// TIA Portal V17 export
// export: Created 2024-09-02T12:50:18.0928197Z, ExportSetting WithDefaults, DisplayName Totally Integrated Automation Portal, DisplayVersion V17, DisplayName TIA Portal Openness, DisplayVersion V17, DisplayName TIA Portal Version Control Interface, DisplayVersion V17, DisplayName STEP 7 Professional, DisplayVersion V17, DisplayName STEP 7 Safety, DisplayVersion V17, DisplayName WinCC Professional, DisplayVersion V17
FUNCTION_BLOCK "LTLL_Main_HMI_OP70"   // FB3, LAD
TITLE = LTLL_HMILite
{ S7_Optimized_Access := 'TRUE' }
AUTHOR : Siemens
FAMILY : HMI_Lite
NAME : LTLL_HMILite
VERSION : 8.10
// stored: AutoNumber true, IsIECCheckEnabled false, IsRetainMemResEnabled false, MemoryReserve 100, SetENOAutomatically false, UDAEnableTagReadback false
   VAR
      instLTLL_Basic { S7_SetPoint := 'True'} : "LTLL_Basic";
      instLTLL_Manual { S7_SetPoint := 'True'} : "LTLL_Manual";
      instLTLL_ManualGraph { S7_SetPoint := 'True'} : "LTLL_ManualGraph";
      instLTLL_Sinamics { S7_SetPoint := 'True'} : "LTLL_Sinamics";
      instLTLL_Motorstarter { S7_SetPoint := 'True'} : "LTLL_Motorstarter";
      instLTLL_RFID { S7_SetPoint := 'True'} : "LTLL_RFID";
      instLTLL_Cycletime_1 { S7_SetPoint := 'True'} : "LTLL_Cycletime";
      instLTLL_Cycletime { S7_SetPoint := 'True'} : "LTLL_Cycletime";
      instLTLL_Counter { S7_SetPoint := 'True'} : "LTLL_Counter";
      instLTLL_PLCSystemData { S7_SetPoint := 'True'} : "LTLL_PLCSystemData";
      instLTLL_Eks { S7_SetPoint := 'True'} : "LTLL_Eks";
   END_VAR
   VAR_TEMP
      tempBasicRetRDSysT : Int;
      tempBasicStatusRDREC : DWord;
      tempBasicStatus : Word;
      tempBasicErrID : Word;
      tempManualStatus : Word;
      tempManualErrID : Word;
      tempManualGraphStatus : Word;
      tempManualGraphErrID : Word;
      tempSinamicsBusy : Bool;
      tempSinamicsStatus : Word;
      tempSinamicsErrID : Word;
      tempSinamicsWrRecStatus : DWord;
      tempSinamicsRdRecStatus : DWord;
      tempMotorstarterBusy : Bool;
      tempMotorstarterRdRec1Status : DWord;
      tempMotorstarterRdRec2Status : DWord;
      tempMotorstarterErrID : Word;
      tempMotorstarterStatus : Word;
      tempRfidStatus : Word;
      tempRfidErrID : Word;
      tempPlcSystemDataStatus : Word;
      tempPlcSystemDataStatusGetImData : Word;
      tempPlcSystemDataErrID : Word;
      tempCounter1Status : Word;
      tempCounter1ErrID : Word;
      tempCycletime1Status : Word;
      tempCycletime1ErrID : Word;
      tempEksProtectionLevel : Int;
      tempEksChecksumNOK : Bool;
      tempEksDateNOK : Bool;
      tempEkscostCenterNOK : Bool;
      tempEksKeyInvalidLess30Days : Bool;
      tempEksAdapterReady : Bool;
      tempEksKeyDetected : Bool;
      tempSchichtReset : Bool;
      tempTagReset : Bool;
      tempZeiger : Int;
      tempAnzGesamt : Int;
      tempAnzNio : Int;
      Cycle_Time_Index : Int;
      t_i : Int;
   END_VAR
   VAR_TEMP   // added for the SCL form of the ladder/FBD networks
      _w1 : Bool;
      _w2 : Bool;
      _w3 : Bool;
   END_VAR
BEGIN

REGION Network 1: Call HMI Lite Basic / Aufruf HMI Lite Basic
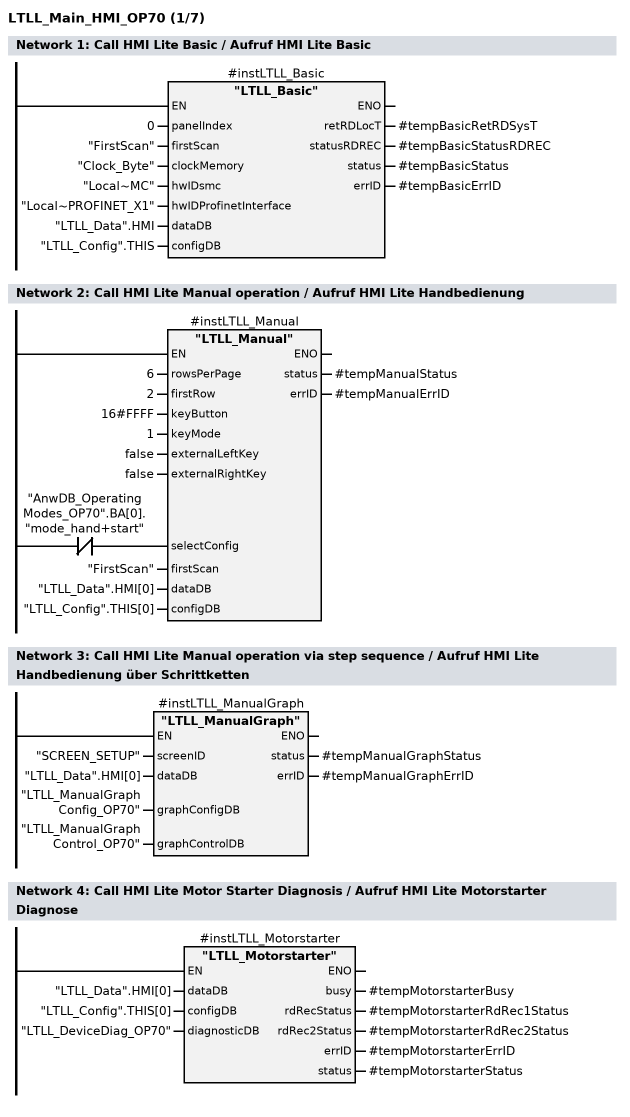
   RUNG wire#powerrail
      #instLTLL_Basic(panelIndex := 0, firstScan := "FirstScan", clockMemory := "Clock_Byte", hwIDsmc := "Local~MC", hwIDProfinetInterface := "Local~PROFINET_X1", dataDB := "LTLL_Data".HMI, configDB := "LTLL_Config".THIS, retRDLocT => #tempBasicRetRDSysT, statusRDREC => #tempBasicStatusRDREC, status => #tempBasicStatus, errID => #tempBasicErrID)
   END_RUNG
   // the same network as SCL:
   #instLTLL_Basic(panelIndex := 0,   // "LTLL_Basic"
                   firstScan := "FirstScan",
                   clockMemory := "Clock_Byte",
                   hwIDsmc := "Local~MC",
                   hwIDProfinetInterface := "Local~PROFINET_X1",
                   dataDB := "LTLL_Data".HMI,
                   configDB := "LTLL_Config".THIS,
                   retRDLocT => #tempBasicRetRDSysT,
                   statusRDREC => #tempBasicStatusRDREC,
                   status => #tempBasicStatus,
                   errID => #tempBasicErrID);
END_REGION

REGION Network 2: Call HMI Lite Manual operation / Aufruf HMI Lite Handbedienung
   RUNG wire#powerrail
      #instLTLL_Manual(selectConfig := wire#w1, rowsPerPage := 6, firstRow := 2, keyButton := 16#FFFF, keyMode := 1, externalLeftKey := false, externalRightKey := false, firstScan := "FirstScan", dataDB := "LTLL_Data".HMI[0], configDB := "LTLL_Config".THIS[0], status => #tempManualStatus, errID => #tempManualErrID)
   END_RUNG
   RUNG wire#powerrail
      I_Contact( "AnwDB_OperatingModes_OP70".BA[0]."mode_hand+start" )
   END_RUNG wire#w1
   // the same network as SCL:
   #instLTLL_Manual(rowsPerPage := 6,   // "LTLL_Manual"
                    firstRow := 2,
                    keyButton := 16#FFFF,
                    keyMode := 1,
                    externalLeftKey := false,
                    externalRightKey := false,
                    selectConfig := NOT "AnwDB_OperatingModes_OP70".BA[0]."mode_hand+start",
                    firstScan := "FirstScan",
                    dataDB := "LTLL_Data".HMI[0],
                    configDB := "LTLL_Config".THIS[0],
                    status => #tempManualStatus,
                    errID => #tempManualErrID);
END_REGION

REGION Network 3: Call HMI Lite Manual operation via step sequence / Aufruf HMI Lite Handbedienung über Schrittketten
   RUNG wire#powerrail
      #instLTLL_ManualGraph(screenID := "SCREEN_SETUP", dataDB := "LTLL_Data".HMI[0], graphConfigDB := "LTLL_ManualGraphConfig_OP70", graphControlDB := "LTLL_ManualGraphControl_OP70", status => #tempManualGraphStatus, errID => #tempManualGraphErrID)
   END_RUNG
   // the same network as SCL:
   #instLTLL_ManualGraph(screenID := "SCREEN_SETUP",   // "LTLL_ManualGraph"
                         dataDB := "LTLL_Data".HMI[0],
                         graphConfigDB := "LTLL_ManualGraphConfig_OP70",
                         graphControlDB := "LTLL_ManualGraphControl_OP70",
                         status => #tempManualGraphStatus,
                         errID => #tempManualGraphErrID);
END_REGION

REGION Network 4: Call HMI Lite Motor Starter Diagnosis / Aufruf HMI Lite Motorstarter Diagnose
   RUNG wire#powerrail
      #instLTLL_Motorstarter(dataDB := "LTLL_Data".HMI[0], configDB := "LTLL_Config".THIS[0], diagnosticDB := "LTLL_DeviceDiag_OP70", busy => #tempMotorstarterBusy, rdRecStatus => #tempMotorstarterRdRec1Status, rdRec2Status => #tempMotorstarterRdRec2Status, errID => #tempMotorstarterErrID, status => #tempMotorstarterStatus)
   END_RUNG
   // the same network as SCL:
   #instLTLL_Motorstarter(dataDB := "LTLL_Data".HMI[0],   // "LTLL_Motorstarter"
                          configDB := "LTLL_Config".THIS[0],
                          diagnosticDB := "LTLL_DeviceDiag_OP70",
                          busy => #tempMotorstarterBusy,
                          rdRecStatus => #tempMotorstarterRdRec1Status,
                          rdRec2Status => #tempMotorstarterRdRec2Status,
                          errID => #tempMotorstarterErrID,
                          status => #tempMotorstarterStatus);
END_REGION

REGION Network 5: Call the HMI Lite RFID Diagnostics / Auruf der HMI Lite RFID Diagnose
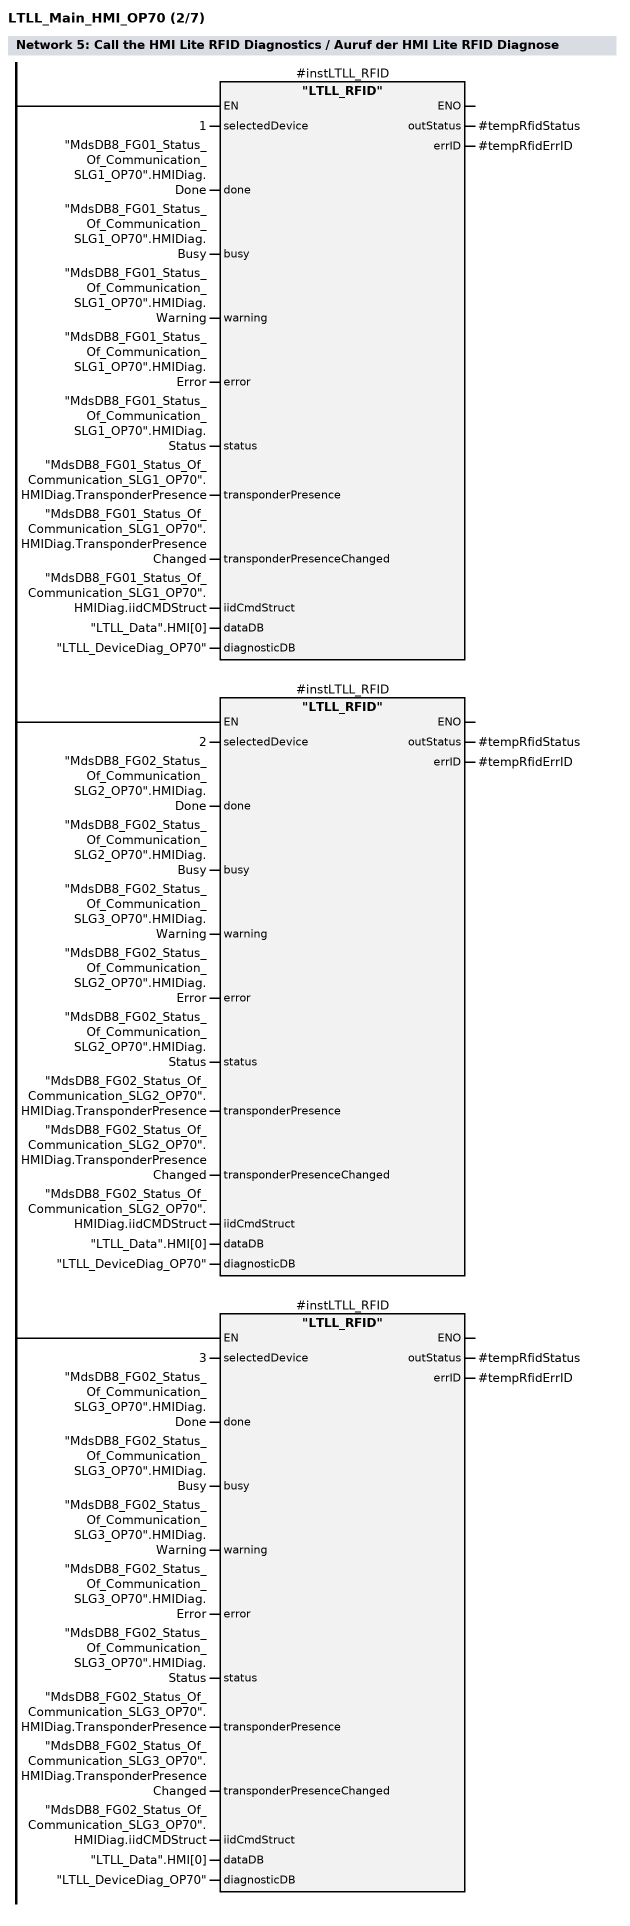
   RUNG wire#powerrail
      #instLTLL_RFID(selectedDevice := 1, done := "MdsDB8_FG01_Status_Of_Communication_SLG1_OP70".HMIDiag.Done, busy := "MdsDB8_FG01_Status_Of_Communication_SLG1_OP70".HMIDiag.Busy, warning := "MdsDB8_FG01_Status_Of_Communication_SLG1_OP70".HMIDiag.Warning, error := "MdsDB8_FG01_Status_Of_Communication_SLG1_OP70".HMIDiag.Error, status := "MdsDB8_FG01_Status_Of_Communication_SLG1_OP70".HMIDiag.Status, transponderPresence := "MdsDB8_FG01_Status_Of_Communication_SLG1_OP70".HMIDiag.TransponderPresence, transponderPresenceChanged := "MdsDB8_FG01_Status_Of_Communication_SLG1_OP70".HMIDiag.TransponderPresenceChanged, iidCmdStruct := "MdsDB8_FG01_Status_Of_Communication_SLG1_OP70".HMIDiag.iidCMDStruct, dataDB := "LTLL_Data".HMI[0], diagnosticDB := "LTLL_DeviceDiag_OP70", outStatus => #tempRfidStatus, errID => #tempRfidErrID)
   END_RUNG
   RUNG wire#powerrail
      #instLTLL_RFID(selectedDevice := 2, done := "MdsDB8_FG02_Status_Of_Communication_SLG2_OP70".HMIDiag.Done, busy := "MdsDB8_FG02_Status_Of_Communication_SLG2_OP70".HMIDiag.Busy, warning := "MdsDB8_FG02_Status_Of_Communication_SLG3_OP70".HMIDiag.Warning, error := "MdsDB8_FG02_Status_Of_Communication_SLG2_OP70".HMIDiag.Error, status := "MdsDB8_FG02_Status_Of_Communication_SLG2_OP70".HMIDiag.Status, transponderPresence := "MdsDB8_FG02_Status_Of_Communication_SLG2_OP70".HMIDiag.TransponderPresence, transponderPresenceChanged := "MdsDB8_FG02_Status_Of_Communication_SLG2_OP70".HMIDiag.TransponderPresenceChanged, iidCmdStruct := "MdsDB8_FG02_Status_Of_Communication_SLG2_OP70".HMIDiag.iidCMDStruct, dataDB := "LTLL_Data".HMI[0], diagnosticDB := "LTLL_DeviceDiag_OP70", outStatus => #tempRfidStatus, errID => #tempRfidErrID)
   END_RUNG
   RUNG wire#powerrail
      #instLTLL_RFID(selectedDevice := 3, done := "MdsDB8_FG02_Status_Of_Communication_SLG3_OP70".HMIDiag.Done, busy := "MdsDB8_FG02_Status_Of_Communication_SLG3_OP70".HMIDiag.Busy, warning := "MdsDB8_FG02_Status_Of_Communication_SLG3_OP70".HMIDiag.Warning, error := "MdsDB8_FG02_Status_Of_Communication_SLG3_OP70".HMIDiag.Error, status := "MdsDB8_FG02_Status_Of_Communication_SLG3_OP70".HMIDiag.Status, transponderPresence := "MdsDB8_FG02_Status_Of_Communication_SLG3_OP70".HMIDiag.TransponderPresence, transponderPresenceChanged := "MdsDB8_FG02_Status_Of_Communication_SLG3_OP70".HMIDiag.TransponderPresenceChanged, iidCmdStruct := "MdsDB8_FG02_Status_Of_Communication_SLG3_OP70".HMIDiag.iidCMDStruct, dataDB := "LTLL_Data".HMI[0], diagnosticDB := "LTLL_DeviceDiag_OP70", outStatus => #tempRfidStatus, errID => #tempRfidErrID)
   END_RUNG
   // the same network as SCL:
   #instLTLL_RFID(selectedDevice := 1,   // "LTLL_RFID"
                  done := "MdsDB8_FG01_Status_Of_Communication_SLG1_OP70".HMIDiag.Done,
                  busy := "MdsDB8_FG01_Status_Of_Communication_SLG1_OP70".HMIDiag.Busy,
                  warning := "MdsDB8_FG01_Status_Of_Communication_SLG1_OP70".HMIDiag.Warning,
                  error := "MdsDB8_FG01_Status_Of_Communication_SLG1_OP70".HMIDiag.Error,
                  status := "MdsDB8_FG01_Status_Of_Communication_SLG1_OP70".HMIDiag.Status,
                  transponderPresence := "MdsDB8_FG01_Status_Of_Communication_SLG1_OP70".HMIDiag.TransponderPresence,
                  transponderPresenceChanged := "MdsDB8_FG01_Status_Of_Communication_SLG1_OP70".HMIDiag.TransponderPresenceChanged,
                  iidCmdStruct := "MdsDB8_FG01_Status_Of_Communication_SLG1_OP70".HMIDiag.iidCMDStruct,
                  dataDB := "LTLL_Data".HMI[0],
                  diagnosticDB := "LTLL_DeviceDiag_OP70",
                  outStatus => #tempRfidStatus,
                  errID => #tempRfidErrID);
   #instLTLL_RFID(selectedDevice := 2,   // "LTLL_RFID"
                  done := "MdsDB8_FG02_Status_Of_Communication_SLG2_OP70".HMIDiag.Done,
                  busy := "MdsDB8_FG02_Status_Of_Communication_SLG2_OP70".HMIDiag.Busy,
                  warning := "MdsDB8_FG02_Status_Of_Communication_SLG3_OP70".HMIDiag.Warning,
                  error := "MdsDB8_FG02_Status_Of_Communication_SLG2_OP70".HMIDiag.Error,
                  status := "MdsDB8_FG02_Status_Of_Communication_SLG2_OP70".HMIDiag.Status,
                  transponderPresence := "MdsDB8_FG02_Status_Of_Communication_SLG2_OP70".HMIDiag.TransponderPresence,
                  transponderPresenceChanged := "MdsDB8_FG02_Status_Of_Communication_SLG2_OP70".HMIDiag.TransponderPresenceChanged,
                  iidCmdStruct := "MdsDB8_FG02_Status_Of_Communication_SLG2_OP70".HMIDiag.iidCMDStruct,
                  dataDB := "LTLL_Data".HMI[0],
                  diagnosticDB := "LTLL_DeviceDiag_OP70",
                  outStatus => #tempRfidStatus,
                  errID => #tempRfidErrID);
   #instLTLL_RFID(selectedDevice := 3,   // "LTLL_RFID"
                  done := "MdsDB8_FG02_Status_Of_Communication_SLG3_OP70".HMIDiag.Done,
                  busy := "MdsDB8_FG02_Status_Of_Communication_SLG3_OP70".HMIDiag.Busy,
                  warning := "MdsDB8_FG02_Status_Of_Communication_SLG3_OP70".HMIDiag.Warning,
                  error := "MdsDB8_FG02_Status_Of_Communication_SLG3_OP70".HMIDiag.Error,
                  status := "MdsDB8_FG02_Status_Of_Communication_SLG3_OP70".HMIDiag.Status,
                  transponderPresence := "MdsDB8_FG02_Status_Of_Communication_SLG3_OP70".HMIDiag.TransponderPresence,
                  transponderPresenceChanged := "MdsDB8_FG02_Status_Of_Communication_SLG3_OP70".HMIDiag.TransponderPresenceChanged,
                  iidCmdStruct := "MdsDB8_FG02_Status_Of_Communication_SLG3_OP70".HMIDiag.iidCMDStruct,
                  dataDB := "LTLL_Data".HMI[0],
                  diagnosticDB := "LTLL_DeviceDiag_OP70",
                  outStatus => #tempRfidStatus,
                  errID => #tempRfidErrID);
END_REGION

REGION Network 6: Call HMI Lite PLC system data / Aufruf HMI Lite PLC Systemdaten
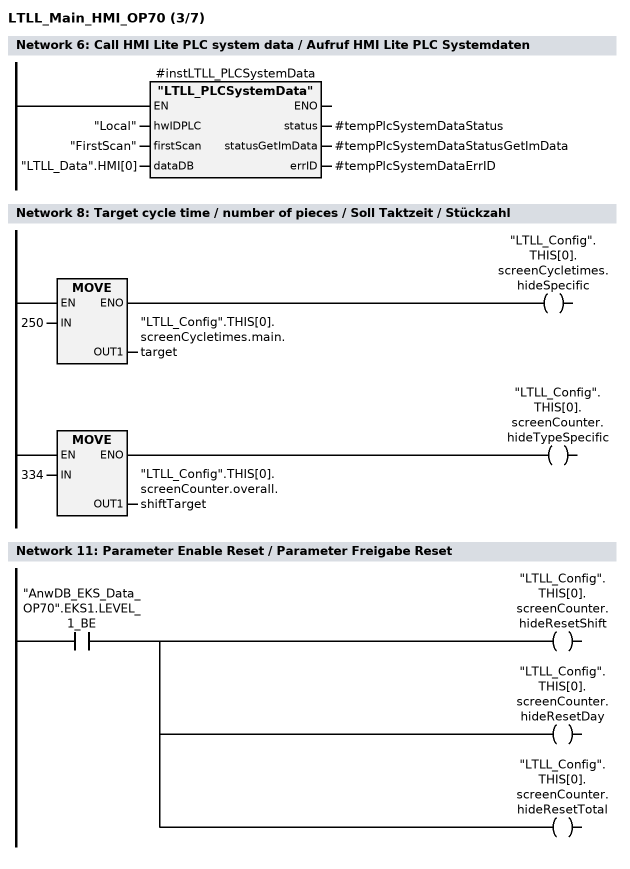
   RUNG wire#powerrail
      #instLTLL_PLCSystemData(hwIDPLC := "Local", firstScan := "FirstScan", dataDB := "LTLL_Data".HMI[0], status => #tempPlcSystemDataStatus, statusGetImData => #tempPlcSystemDataStatusGetImData, errID => #tempPlcSystemDataErrID)
   END_RUNG
   // the same network as SCL:
   #instLTLL_PLCSystemData(hwIDPLC := "Local",   // "LTLL_PLCSystemData"
                           firstScan := "FirstScan",
                           dataDB := "LTLL_Data".HMI[0],
                           status => #tempPlcSystemDataStatus,
                           statusGetImData => #tempPlcSystemDataStatusGetImData,
                           errID => #tempPlcSystemDataErrID);
END_REGION

REGION Network 7: Call HMI Lite Safety Diagnosis / Aufruf HMI Lite Safety Diagnose
END_REGION

REGION Network 8: Target cycle time / number of pieces / Soll Taktzeit / Stückzahl
   RUNG wire#powerrail
      Move(in := 250, out1 => "LTLL_Config".THIS[0].screenCycletimes.main.target)
      Coil( "LTLL_Config".THIS[0].screenCycletimes.hideSpecific )
   END_RUNG
   RUNG wire#powerrail
      Move(in := 334, out1 => "LTLL_Config".THIS[0].screenCounter.overall.shiftTarget)
      Coil( "LTLL_Config".THIS[0].screenCounter.hideTypeSpecific )
   END_RUNG
   // the same network as SCL:
   "LTLL_Config".THIS[0].screenCycletimes.main.target := 250;
   "LTLL_Config".THIS[0].screenCycletimes.hideSpecific := TRUE;
   "LTLL_Config".THIS[0].screenCounter.overall.shiftTarget := 334;
   "LTLL_Config".THIS[0].screenCounter.hideTypeSpecific := TRUE;
END_REGION

REGION Network 9 (SCL): Target cycle time Sub
   FOR #t_i := 0 TO 14 DO
       "LTLL_Config".THIS[0].screenCycletimes.sub.target[#t_i] := "LTLL_Config".THIS[0].screenCycletimes.main.target;

   END_FOR;
END_REGION

REGION Network 10 (SCL): Specific quantity Target quantity / Stückzahl spezifisch Soll
   FOR #tempZeiger := 0 TO 31 DO
       "LTLL_CounterData_OP70".specific[#tempZeiger].config.shiftTarget := 0;
   END_FOR;
END_REGION

REGION Network 11: Parameter Enable Reset / Parameter Freigabe Reset
   RUNG wire#powerrail
      Contact( "AnwDB_EKS_Data_OP70".EKS1.LEVEL_1_BE )
      wire#w1
      Coil( "LTLL_Config".THIS[0].screenCounter.hideResetShift )
   END_RUNG
   RUNG wire#w1
      Coil( "LTLL_Config".THIS[0].screenCounter.hideResetDay )
   END_RUNG
   RUNG wire#w1
      Coil( "LTLL_Config".THIS[0].screenCounter.hideResetTotal )
   END_RUNG
   // the same network as SCL:
   "LTLL_Config".THIS[0].screenCounter.hideResetShift := "AnwDB_EKS_Data_OP70".EKS1.LEVEL_1_BE;
   "LTLL_Config".THIS[0].screenCounter.hideResetDay := "AnwDB_EKS_Data_OP70".EKS1.LEVEL_1_BE;
   "LTLL_Config".THIS[0].screenCounter.hideResetTotal := "AnwDB_EKS_Data_OP70".EKS1.LEVEL_1_BE;
END_REGION

REGION Network 12: Quantity Reset / Stückzahl Reset
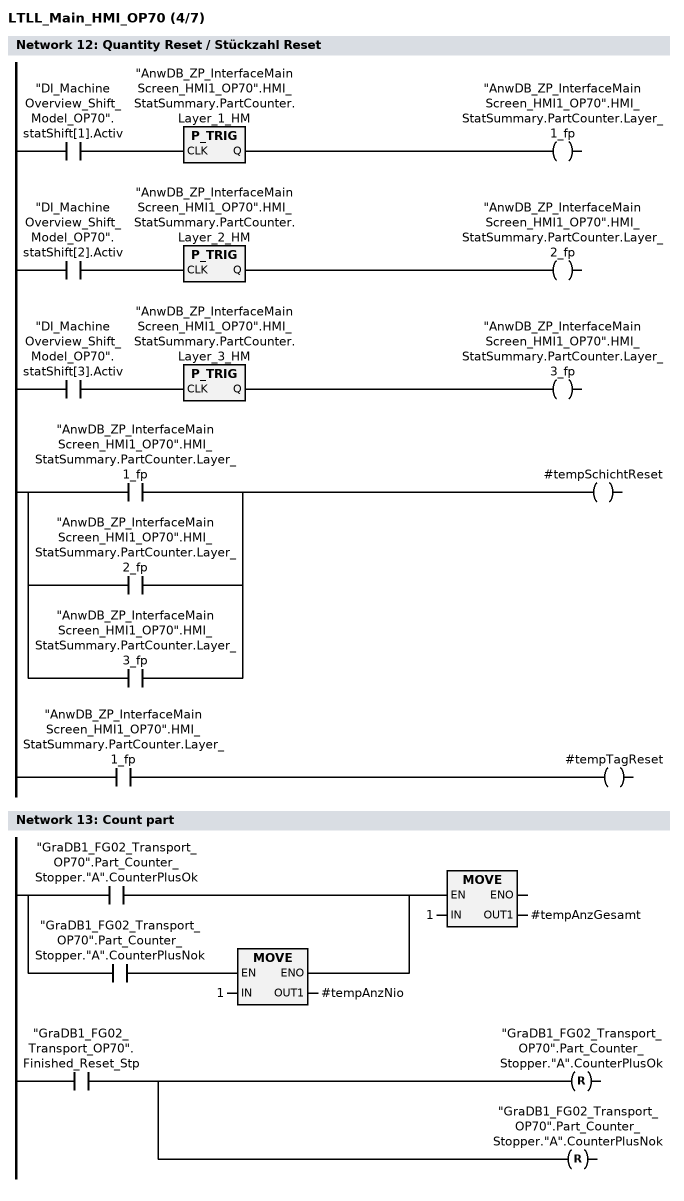
   RUNG wire#powerrail
      Contact( "DI_MachineOverview_Shift_Model_OP70".statShift[1].Activ )
      P_Trig( "AnwDB_ZP_InterfaceMainScreen_HMI1_OP70".HMI_StatSummary.PartCounter.Layer_1_HM )
      Coil( "AnwDB_ZP_InterfaceMainScreen_HMI1_OP70".HMI_StatSummary.PartCounter.Layer_1_fp )
   END_RUNG
   RUNG wire#powerrail
      Contact( "DI_MachineOverview_Shift_Model_OP70".statShift[2].Activ )
      P_Trig( "AnwDB_ZP_InterfaceMainScreen_HMI1_OP70".HMI_StatSummary.PartCounter.Layer_2_HM )
      Coil( "AnwDB_ZP_InterfaceMainScreen_HMI1_OP70".HMI_StatSummary.PartCounter.Layer_2_fp )
   END_RUNG
   RUNG wire#powerrail
      Contact( "DI_MachineOverview_Shift_Model_OP70".statShift[3].Activ )
      P_Trig( "AnwDB_ZP_InterfaceMainScreen_HMI1_OP70".HMI_StatSummary.PartCounter.Layer_3_HM )
      Coil( "AnwDB_ZP_InterfaceMainScreen_HMI1_OP70".HMI_StatSummary.PartCounter.Layer_3_fp )
   END_RUNG
   RUNG wire#powerrail
      Contact( "AnwDB_ZP_InterfaceMainScreen_HMI1_OP70".HMI_StatSummary.PartCounter.Layer_1_fp )
      wire#w1
      Coil( #tempSchichtReset )
   END_RUNG
   RUNG wire#powerrail
      Contact( "AnwDB_ZP_InterfaceMainScreen_HMI1_OP70".HMI_StatSummary.PartCounter.Layer_2_fp )
   END_RUNG wire#w1
   RUNG wire#powerrail
      Contact( "AnwDB_ZP_InterfaceMainScreen_HMI1_OP70".HMI_StatSummary.PartCounter.Layer_3_fp )
   END_RUNG wire#w1
   RUNG wire#powerrail
      Contact( "AnwDB_ZP_InterfaceMainScreen_HMI1_OP70".HMI_StatSummary.PartCounter.Layer_1_fp )
      Coil( #tempTagReset )
   END_RUNG
   // the same network as SCL:
   #_w1 := "DI_MachineOverview_Shift_Model_OP70".statShift[1].Activ AND NOT "AnwDB_ZP_InterfaceMainScreen_HMI1_OP70".HMI_StatSummary.PartCounter.Layer_1_HM;   // rising edge
   "AnwDB_ZP_InterfaceMainScreen_HMI1_OP70".HMI_StatSummary.PartCounter.Layer_1_HM := "DI_MachineOverview_Shift_Model_OP70".statShift[1].Activ;
   "AnwDB_ZP_InterfaceMainScreen_HMI1_OP70".HMI_StatSummary.PartCounter.Layer_1_fp := #_w1;
   #_w2 := "DI_MachineOverview_Shift_Model_OP70".statShift[2].Activ AND NOT "AnwDB_ZP_InterfaceMainScreen_HMI1_OP70".HMI_StatSummary.PartCounter.Layer_2_HM;   // rising edge
   "AnwDB_ZP_InterfaceMainScreen_HMI1_OP70".HMI_StatSummary.PartCounter.Layer_2_HM := "DI_MachineOverview_Shift_Model_OP70".statShift[2].Activ;
   "AnwDB_ZP_InterfaceMainScreen_HMI1_OP70".HMI_StatSummary.PartCounter.Layer_2_fp := #_w2;
   #_w3 := "DI_MachineOverview_Shift_Model_OP70".statShift[3].Activ AND NOT "AnwDB_ZP_InterfaceMainScreen_HMI1_OP70".HMI_StatSummary.PartCounter.Layer_3_HM;   // rising edge
   "AnwDB_ZP_InterfaceMainScreen_HMI1_OP70".HMI_StatSummary.PartCounter.Layer_3_HM := "DI_MachineOverview_Shift_Model_OP70".statShift[3].Activ;
   "AnwDB_ZP_InterfaceMainScreen_HMI1_OP70".HMI_StatSummary.PartCounter.Layer_3_fp := #_w3;
   #tempSchichtReset := "AnwDB_ZP_InterfaceMainScreen_HMI1_OP70".HMI_StatSummary.PartCounter.Layer_1_fp OR "AnwDB_ZP_InterfaceMainScreen_HMI1_OP70".HMI_StatSummary.PartCounter.Layer_2_fp OR "AnwDB_ZP_InterfaceMainScreen_HMI1_OP70".HMI_StatSummary.PartCounter.Layer_3_fp;
   #tempTagReset := "AnwDB_ZP_InterfaceMainScreen_HMI1_OP70".HMI_StatSummary.PartCounter.Layer_1_fp;
END_REGION

REGION Network 13: Count part
   RUNG wire#powerrail
      Contact( "GraDB1_FG02_Transport_OP70".Part_Counter_Stopper."A".CounterPlusOk )
      wire#w1
      Move(in := 1, out1 => #tempAnzGesamt)
   END_RUNG
   RUNG wire#powerrail
      Contact( "GraDB1_FG02_Transport_OP70".Part_Counter_Stopper."A".CounterPlusNok )
      Move(in := 1, out1 => #tempAnzNio)
   END_RUNG wire#w1
   RUNG wire#powerrail
      Contact( "GraDB1_FG02_Transport_OP70".Finished_Reset_Stp )
      wire#w2
      R_Coil( "GraDB1_FG02_Transport_OP70".Part_Counter_Stopper."A".CounterPlusOk )
   END_RUNG
   RUNG wire#w2
      R_Coil( "GraDB1_FG02_Transport_OP70".Part_Counter_Stopper."A".CounterPlusNok )
   END_RUNG
   // the same network as SCL:
   IF "GraDB1_FG02_Transport_OP70".Part_Counter_Stopper."A".CounterPlusNok THEN #tempAnzNio := 1; END_IF;
   IF "GraDB1_FG02_Transport_OP70".Part_Counter_Stopper."A".CounterPlusOk OR "GraDB1_FG02_Transport_OP70".Part_Counter_Stopper."A".CounterPlusNok THEN
       #tempAnzGesamt := 1;
   END_IF;
   IF "GraDB1_FG02_Transport_OP70".Finished_Reset_Stp THEN
       "GraDB1_FG02_Transport_OP70".Part_Counter_Stopper."A".CounterPlusOk := FALSE;
       "GraDB1_FG02_Transport_OP70".Part_Counter_Stopper."A".CounterPlusNok := FALSE;
   END_IF;
END_REGION

REGION Network 14: Call HMI Lite piece counter / Aufruf HMI Lite Stückzähler
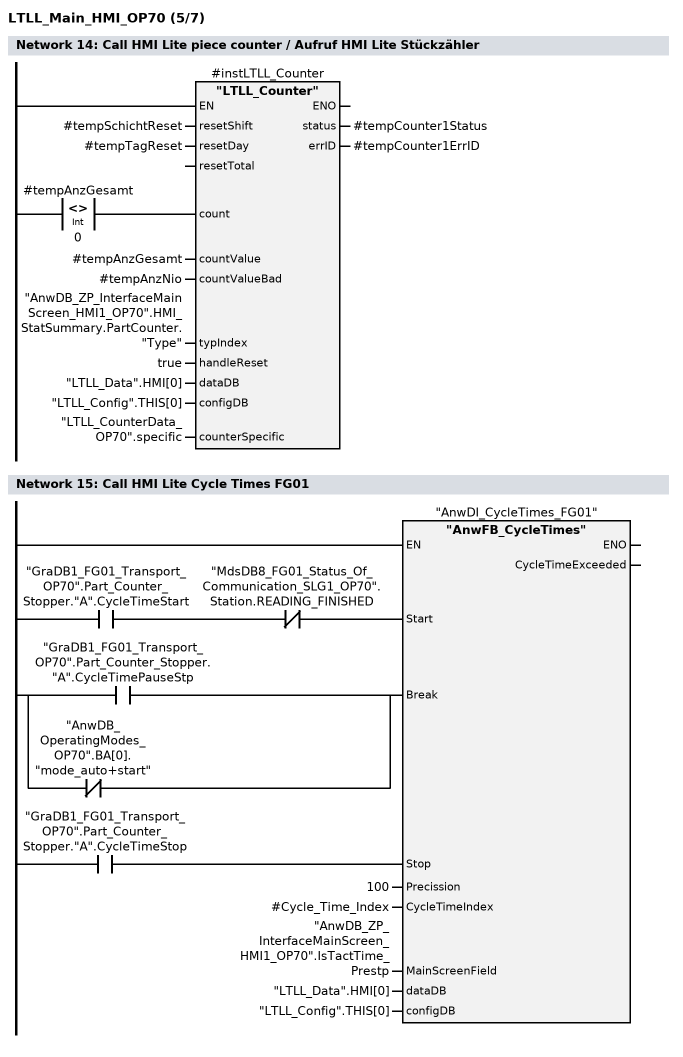
   RUNG wire#powerrail
      #instLTLL_Counter(count := wire#w1, resetShift := #tempSchichtReset, resetDay := #tempTagReset, resetTotal :=, countValue := #tempAnzGesamt, countValueBad := #tempAnzNio, typIndex := "AnwDB_ZP_InterfaceMainScreen_HMI1_OP70".HMI_StatSummary.PartCounter."Type", handleReset := true, dataDB := "LTLL_Data".HMI[0], configDB := "LTLL_Config".THIS[0], counterSpecific := "LTLL_CounterData_OP70".specific, status => #tempCounter1Status, errID => #tempCounter1ErrID)
   END_RUNG
   RUNG wire#powerrail
      { S7_Templates := "SrcType := Int" } NE_Contact(in1 := #tempAnzGesamt, in2 := 0)
   END_RUNG wire#w1
   // the same network as SCL:
   #instLTLL_Counter(resetShift := #tempSchichtReset,   // "LTLL_Counter"
                     resetDay := #tempTagReset,
                     count := #tempAnzGesamt <> 0,
                     countValue := #tempAnzGesamt,
                     countValueBad := #tempAnzNio,
                     typIndex := "AnwDB_ZP_InterfaceMainScreen_HMI1_OP70".HMI_StatSummary.PartCounter."Type",
                     handleReset := true,
                     dataDB := "LTLL_Data".HMI[0],
                     configDB := "LTLL_Config".THIS[0],
                     counterSpecific := "LTLL_CounterData_OP70".specific,
                     status => #tempCounter1Status,
                     errID => #tempCounter1ErrID);
END_REGION

REGION Network 15: Call HMI Lite Cycle Times FG01
   RUNG wire#powerrail
      "AnwDI_CycleTimes_FG01"(Start := wire#w1, Break := wire#w2, Stop := wire#w3, Precission := 100, CycleTimeIndex := #Cycle_Time_Index, MainScreenField := "AnwDB_ZP_InterfaceMainScreen_HMI1_OP70".IsTactTime_Prestp, dataDB := "LTLL_Data".HMI[0], configDB := "LTLL_Config".THIS[0], CycleTimeExceeded =>)
   END_RUNG
   RUNG wire#powerrail
      Contact( "GraDB1_FG01_Transport_OP70".Part_Counter_Stopper."A".CycleTimeStart )
      I_Contact( "MdsDB8_FG01_Status_Of_Communication_SLG1_OP70".Station.READING_FINISHED )
   END_RUNG wire#w1
   RUNG wire#powerrail
      Contact( "GraDB1_FG01_Transport_OP70".Part_Counter_Stopper."A".CycleTimePauseStp )
   END_RUNG wire#w2
   RUNG wire#powerrail
      I_Contact( "AnwDB_OperatingModes_OP70".BA[0]."mode_auto+start" )
   END_RUNG wire#w2
   RUNG wire#powerrail
      Contact( "GraDB1_FG01_Transport_OP70".Part_Counter_Stopper."A".CycleTimeStop )
   END_RUNG wire#w3
   // the same network as SCL:
   "AnwDI_CycleTimes_FG01"(Start := "GraDB1_FG01_Transport_OP70".Part_Counter_Stopper."A".CycleTimeStart AND NOT "MdsDB8_FG01_Status_Of_Communication_SLG1_OP70".Station.READING_FINISHED,   // "AnwFB_CycleTimes"
                           Break := "GraDB1_FG01_Transport_OP70".Part_Counter_Stopper."A".CycleTimePauseStp OR NOT "AnwDB_OperatingModes_OP70".BA[0]."mode_auto+start",
                           Stop := "GraDB1_FG01_Transport_OP70".Part_Counter_Stopper."A".CycleTimeStop,
                           Precission := 100,
                           CycleTimeIndex := #Cycle_Time_Index,
                           MainScreenField := "AnwDB_ZP_InterfaceMainScreen_HMI1_OP70".IsTactTime_Prestp,
                           dataDB := "LTLL_Data".HMI[0],
                           configDB := "LTLL_Config".THIS[0]);
END_REGION

REGION Network 16: Call HMI Lite Cycle Times FG02
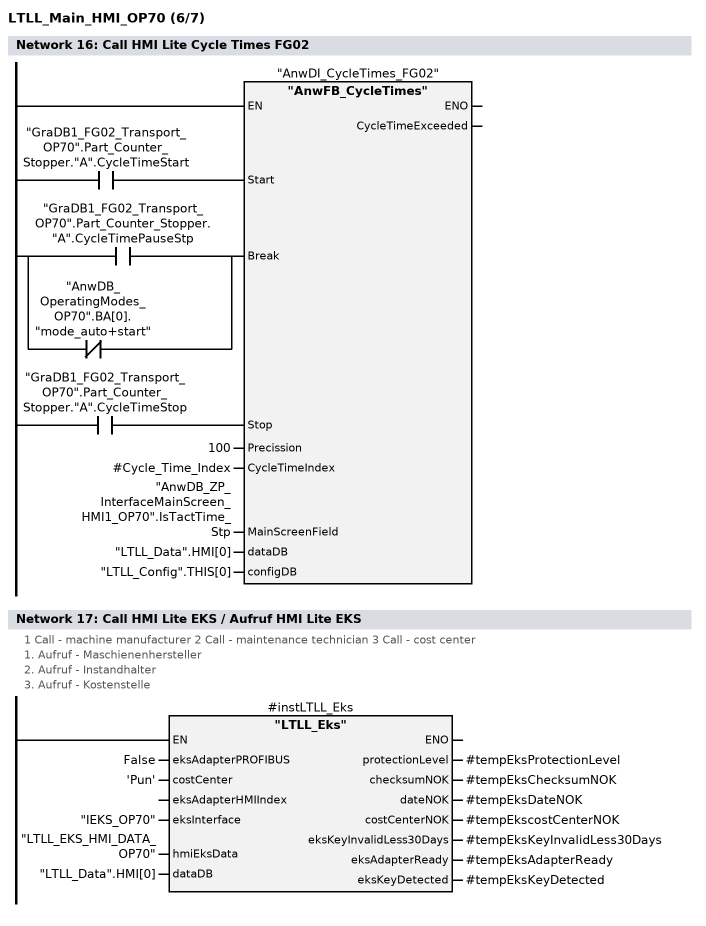
   RUNG wire#powerrail
      "AnwDI_CycleTimes_FG02"(Start := wire#w1, Break := wire#w2, Stop := wire#w3, Precission := 100, CycleTimeIndex := #Cycle_Time_Index, MainScreenField := "AnwDB_ZP_InterfaceMainScreen_HMI1_OP70".IsTactTime_Stp, dataDB := "LTLL_Data".HMI[0], configDB := "LTLL_Config".THIS[0], CycleTimeExceeded =>)
   END_RUNG
   RUNG wire#powerrail
      Contact( "GraDB1_FG02_Transport_OP70".Part_Counter_Stopper."A".CycleTimeStart )
   END_RUNG wire#w1
   RUNG wire#powerrail
      Contact( "GraDB1_FG02_Transport_OP70".Part_Counter_Stopper."A".CycleTimePauseStp )
   END_RUNG wire#w2
   RUNG wire#powerrail
      I_Contact( "AnwDB_OperatingModes_OP70".BA[0]."mode_auto+start" )
   END_RUNG wire#w2
   RUNG wire#powerrail
      Contact( "GraDB1_FG02_Transport_OP70".Part_Counter_Stopper."A".CycleTimeStop )
   END_RUNG wire#w3
   // the same network as SCL:
   "AnwDI_CycleTimes_FG02"(Start := "GraDB1_FG02_Transport_OP70".Part_Counter_Stopper."A".CycleTimeStart,   // "AnwFB_CycleTimes"
                           Break := "GraDB1_FG02_Transport_OP70".Part_Counter_Stopper."A".CycleTimePauseStp OR NOT "AnwDB_OperatingModes_OP70".BA[0]."mode_auto+start",
                           Stop := "GraDB1_FG02_Transport_OP70".Part_Counter_Stopper."A".CycleTimeStop,
                           Precission := 100,
                           CycleTimeIndex := #Cycle_Time_Index,
                           MainScreenField := "AnwDB_ZP_InterfaceMainScreen_HMI1_OP70".IsTactTime_Stp,
                           dataDB := "LTLL_Data".HMI[0],
                           configDB := "LTLL_Config".THIS[0]);
END_REGION

REGION Network 17: Call HMI Lite EKS / Aufruf HMI Lite EKS
   // 1 Call - machine manufacturer 2 Call - maintenance technician 3 Call - cost center
   // 1. Aufruf - Maschienenhersteller
   // 2. Aufruf - Instandhalter
   // 3. Aufruf - Kostenstelle
   RUNG wire#powerrail
      #instLTLL_Eks(eksAdapterPROFIBUS := False, costCenter := 'Pun', eksAdapterHMIIndex :=, eksInterface := "IEKS_OP70", hmiEksData := "LTLL_EKS_HMI_DATA_OP70", dataDB := "LTLL_Data".HMI[0], protectionLevel => #tempEksProtectionLevel, checksumNOK => #tempEksChecksumNOK, dateNOK => #tempEksDateNOK, costCenterNOK => #tempEkscostCenterNOK, eksKeyInvalidLess30Days => #tempEksKeyInvalidLess30Days, eksAdapterReady => #tempEksAdapterReady, eksKeyDetected => #tempEksKeyDetected)
   END_RUNG
   // the same network as SCL:
   #instLTLL_Eks(eksAdapterPROFIBUS := False,   // "LTLL_Eks"
                 costCenter := 'Pun',
                 eksInterface := "IEKS_OP70",
                 hmiEksData := "LTLL_EKS_HMI_DATA_OP70",
                 dataDB := "LTLL_Data".HMI[0],
                 protectionLevel => #tempEksProtectionLevel,
                 checksumNOK => #tempEksChecksumNOK,
                 dateNOK => #tempEksDateNOK,
                 costCenterNOK => #tempEkscostCenterNOK,
                 eksKeyInvalidLess30Days => #tempEksKeyInvalidLess30Days,
                 eksAdapterReady => #tempEksAdapterReady,
                 eksKeyDetected => #tempEksKeyDetected);
END_REGION

REGION Network 18: Protection Level 1 - Red Administrator (Level 1) / Schutzstufe 1 - Rot Administrator (Level 1)
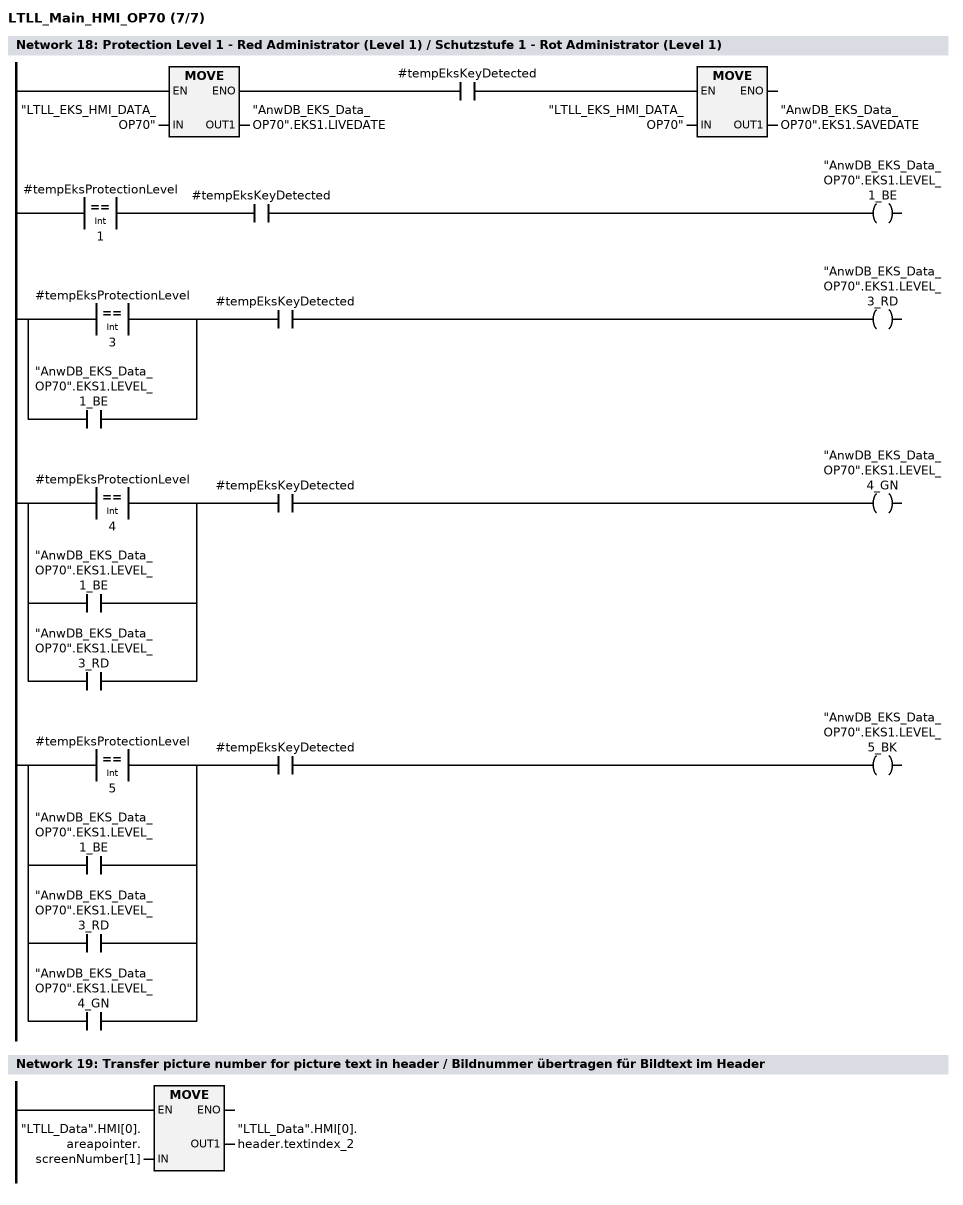
   RUNG wire#powerrail
      Move(in := "LTLL_EKS_HMI_DATA_OP70", out1 => "AnwDB_EKS_Data_OP70".EKS1.LIVEDATE)
      Contact( #tempEksKeyDetected )
      Move(in := "LTLL_EKS_HMI_DATA_OP70", out1 => "AnwDB_EKS_Data_OP70".EKS1.SAVEDATE)
   END_RUNG
   RUNG wire#powerrail
      { S7_Templates := "SrcType := Int" } EQ_Contact(in1 := #tempEksProtectionLevel, in2 := 1)
      Contact( #tempEksKeyDetected )
      Coil( "AnwDB_EKS_Data_OP70".EKS1.LEVEL_1_BE )
   END_RUNG
   RUNG wire#powerrail
      { S7_Templates := "SrcType := Int" } EQ_Contact(in1 := #tempEksProtectionLevel, in2 := 3)
      wire#w1
      Contact( #tempEksKeyDetected )
      Coil( "AnwDB_EKS_Data_OP70".EKS1.LEVEL_3_RD )
   END_RUNG
   RUNG wire#powerrail
      Contact( "AnwDB_EKS_Data_OP70".EKS1.LEVEL_1_BE )
   END_RUNG wire#w1
   RUNG wire#powerrail
      { S7_Templates := "SrcType := Int" } EQ_Contact(in1 := #tempEksProtectionLevel, in2 := 4)
      wire#w2
      Contact( #tempEksKeyDetected )
      Coil( "AnwDB_EKS_Data_OP70".EKS1.LEVEL_4_GN )
   END_RUNG
   RUNG wire#powerrail
      Contact( "AnwDB_EKS_Data_OP70".EKS1.LEVEL_1_BE )
   END_RUNG wire#w2
   RUNG wire#powerrail
      Contact( "AnwDB_EKS_Data_OP70".EKS1.LEVEL_3_RD )
   END_RUNG wire#w2
   RUNG wire#powerrail
      { S7_Templates := "SrcType := Int" } EQ_Contact(in1 := #tempEksProtectionLevel, in2 := 5)
      wire#w3
      Contact( #tempEksKeyDetected )
      Coil( "AnwDB_EKS_Data_OP70".EKS1.LEVEL_5_BK )
   END_RUNG
   RUNG wire#powerrail
      Contact( "AnwDB_EKS_Data_OP70".EKS1.LEVEL_1_BE )
   END_RUNG wire#w3
   RUNG wire#powerrail
      Contact( "AnwDB_EKS_Data_OP70".EKS1.LEVEL_3_RD )
   END_RUNG wire#w3
   RUNG wire#powerrail
      Contact( "AnwDB_EKS_Data_OP70".EKS1.LEVEL_4_GN )
   END_RUNG wire#w3
   // the same network as SCL:
   "AnwDB_EKS_Data_OP70".EKS1.LIVEDATE := "LTLL_EKS_HMI_DATA_OP70";
   IF #tempEksKeyDetected THEN "AnwDB_EKS_Data_OP70".EKS1.SAVEDATE := "LTLL_EKS_HMI_DATA_OP70"; END_IF;
   "AnwDB_EKS_Data_OP70".EKS1.LEVEL_1_BE := (#tempEksProtectionLevel = 1) AND #tempEksKeyDetected;
   "AnwDB_EKS_Data_OP70".EKS1.LEVEL_3_RD := ((#tempEksProtectionLevel = 3) OR "AnwDB_EKS_Data_OP70".EKS1.LEVEL_1_BE) AND #tempEksKeyDetected;
   "AnwDB_EKS_Data_OP70".EKS1.LEVEL_4_GN := ((#tempEksProtectionLevel = 4) OR "AnwDB_EKS_Data_OP70".EKS1.LEVEL_1_BE OR "AnwDB_EKS_Data_OP70".EKS1.LEVEL_3_RD) AND #tempEksKeyDetected;
   "AnwDB_EKS_Data_OP70".EKS1.LEVEL_5_BK := ((#tempEksProtectionLevel = 5) OR "AnwDB_EKS_Data_OP70".EKS1.LEVEL_1_BE OR "AnwDB_EKS_Data_OP70".EKS1.LEVEL_3_RD OR "AnwDB_EKS_Data_OP70".EKS1.LEVEL_4_GN) AND #tempEksKeyDetected;
END_REGION

REGION Network 19: Transfer picture number for picture text in header / Bildnummer übertragen für Bildtext im Header
   RUNG wire#powerrail
      { S7_GenerateENO := "TRUE" } Move(in := "LTLL_Data".HMI[0].areapointer.screenNumber[1], out1 => "LTLL_Data".HMI[0].header.textindex_2)
   END_RUNG
   // the same network as SCL:
   "LTLL_Data".HMI[0].header.textindex_2 := "LTLL_Data".HMI[0].areapointer.screenNumber[1];
END_REGION
END_FUNCTION_BLOCK
